{attribute addProperty BoxType "EL5151-0080-0016"}
{attribute addProperty Id "Enable_latch_CAT %Q*BOOL811Enable_latch_extern_on_positive_edgeAT %Q*BOOL812Set_counterAT %Q*BOOL813Enable_latch_extern_on_negative_edgeAT %Q*BOOL814Set_counter_valueAT %Q*UINT16217"}
{attribute addProperty CRC "2917873719"}
{attribute addProperty SizeInBites "48"}
{attribute addProperty SizeInBytes "6"}
TYPE ENC_Outputs_ADEB3837 :
STRUCT
	{attribute addProperty Name "Enable_latch_C"}
	Enable_latch_C AT %Q* : BOOL;
	{attribute addProperty Name "Enable_latch_extern_on_positive_edge"}
	Enable_latch_extern_on_positive_edge AT %Q* : BOOL;
	{attribute addProperty Name "Set_counter"}
	Set_counter AT %Q* : BOOL;
	{attribute addProperty Name "Enable_latch_extern_on_negative_edge"}
	Enable_latch_extern_on_negative_edge AT %Q* : BOOL;
	{attribute addProperty Name "Set_counter_value"}
	Set_counter_value AT %Q* : UINT;
END_STRUCT
END_TYPE

(* stored: Version 1.2.0.0, ProductVersion 3.1.4024.9
   DUT ENC_Outputs_ADEB3837: Id {a108b54a-f9e5-409f-b6d1-93ef62e07d8c} *)
